TYPE
    TcoTransferSystem_Config EXTENDS TcoCore.TcoStruct :
    STRUCT
     	InfoTime : TIME := T#5S;
        ErrorTime : TIME := T#0S;
        StabilisationTime : TIME := T#200MS;
		HasPositionUnit : BOOL :=TRUE;
		
    END_STRUCT
END_TYPE

(* stored: Version 1.1.0.1
   DUT TcoTransferSystem_Config: Id {aaf0c867-0085-4d82-ac83-276020cec609} *)
